// LS Electric XG5000 project: 1_2INV_단자대운전_정역정지인터록제어_직접제어
// PLC NewPLC

PROGRAM Test_Program_1 (task: 스캔 프로그램)

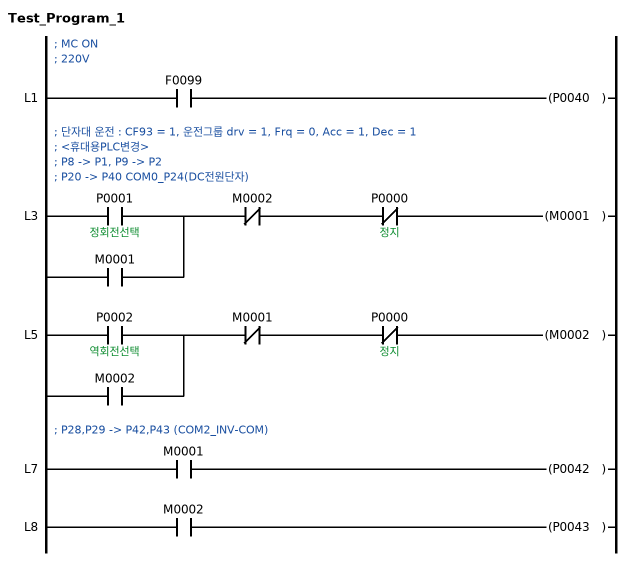
// MC ON
; L1
LOAD      F0099
OUT       P0040
// output comment: 220V
// 단자대 운전 : CF93 = 1, 운전그룹 drv = 1, Frq = 0, Acc = 1, Dec = 1
; L3
LOAD      P0001	// 정회전선택
OR        M0001
AND NOT   M0002
AND NOT   P0000	// 정지
OUT       M0001
// output comment: <휴대용PLC변경>  P8 -> P1, P9 -> P2  P20 -> P40 COM0_P24(DC전원단자)
; L5
LOAD      P0002	// 역회전선택
OR        M0002
AND NOT   M0001
AND NOT   P0000	// 정지
OUT       M0002
; L7
LOAD      M0001
OUT       P0042
// output comment: P28,P29 -> P42,P43 (COM2_INV-COM)
; L8
LOAD      M0002
OUT       P0043

VARIABLES AND COMMENTS (devices not used above)
P00003	BIT	기동
P00007	BIT	역회전
P00006	BIT	정회전